// TIA Portal V19 export
TYPE "LSNTP_typeTimestamp"
// stored: Access Published
   STRUCT
      sec : DWord;   // Time in seconds since 1900-01-01-00:00:00
      secFrac : DWord;   // Fraction of the current second
   END_STRUCT;
END_TYPE
